// TIA Portal V20 export
TYPE "typeCmControlNode"
// stored: Namespace Unit1.Em5
   STRUCT
      Interlock { ExternalWritable := 'False'} : "Unit1.Em5.typeCmControlNodeInterlock";
      softcam { ExternalWritable := 'False'} : "Unit1.Em5.typeCmControlNodeSoftCam";
      brakeTest { ExternalWritable := 'False'} : "Unit1.Em5.typeCmControlNodeBrakeTest";
   END_STRUCT;
END_TYPE
